// TIA Portal V16 export
// export: Created 2021-09-08T12:46:15.0127736Z, ExportSetting WithDefaults, DisplayName Totally Integrated Automation Portal, DisplayVersion V16 Update 3, DisplayName TIA Portal Version Control Interface, DisplayVersion V16 Update 2, DisplayName TIA Portal Openness, DisplayVersion V16 Update 3, DisplayName TIA Portal Teamcenter Gateway, DisplayVersion V16, DisplayName STEP 7 Professional, DisplayVersion V16 Update 3, DisplayName STEP 7 Safety, DisplayVersion V16, DisplayName WinCC Advanced, DisplayVersion V16 Update 3
DATA_BLOCK "AllUfParam_DB"   // DB30
VERSION : 0.1
// stored: AutoNumber true, DBAccessibleFromOPCUA true, InstanceOfName AllUfParam, InstanceOfType FB
"AllUfParam"
   // VAR
   //    mSec : USInt;
   //    sec : UInt;
   //    inVolumeUF1 : Real;
   //    inVolumeUF2 : Real;
   //    outVolumeUF1 : Real;
   //    outVolumeUF2 : Real;
   // END_VAR
BEGIN
END_DATA_BLOCK
